(* Logix 5000 project; controller Drives_Line1 1756-L72 rev 20.13; software revision 20.04; part 16 of 21 *)
(* tags used below, declared in another part *)
   Exit_Accu_FBCounts_mm : DINT;
   Exit_Accu_Rev_mm : REAL;
   IO_State_Exit_Accu : INT;
   IO_State_Tmp_Exit_Accu : INT;
   ons : BOOL[32];
   TofReset : TIMER;
   TonNoResponse : TIMER;
   TonRefOn : TIMER;
   TonTensionOnSp : TIMER;
   zExit_Accu_EncCounts : DINT;
   zExit_Accu_Kp_Preg : REAL;
   zExit_Accu_Kp_Treg : REAL;
   zExit_Accu_MaxAccDec : REAL;
   zExit_Accu_NrOfCyl : DINT;
   zExit_Accu_Pos_PreLim : REAL;
   zExit_Accu_SpdRegMax : REAL;
   zExit_Accu_SpdRegMin : REAL;
   zExit_Accu_SpdTrim_HL : REAL;
   zExit_Accu_SpdtRim_LL : REAL;
   zExit_Accu_WLD_Preg : REAL;
   zExit_Accu_WLD_Treg : REAL;
   zNoMaster : BOOL;
   zTM3_Tens_Offset : REAL;
   Bridle_04 : UDT_Bridle_3M;
   EntryConfig : UDT_Config_Zone;
   Exit_Accu : UDT_Exit_Accu;
   ExitConfig : UDT_Config_Zone;
   ExitCtrl : UDT_Control_Zone;
   ExitStat : UDT_Status_Zone;
   In_Commands : UDT_Commands;
   In_Config : UDT_Config;
   In_Setpoints : UDT_Setpoints;
   LineCmd : UDT_Commands_Line;
   LineCtrl : UDT_Control_Line;
   LineStat : UDT_Status_Line;
   TM3 : UDT_TM;
(* P18_Exit_Accu, continued *)

ROUTINE R01_From_Master   (* ladder *)
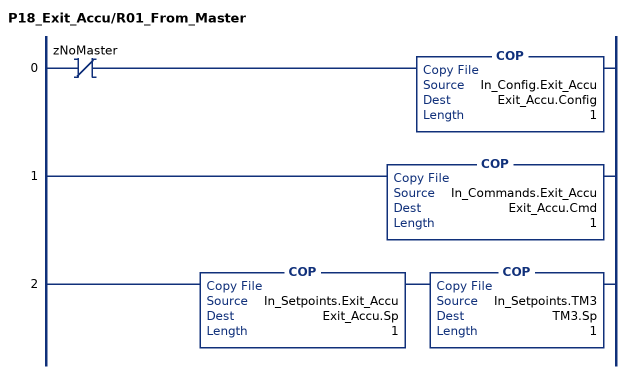
   0: XIO(zNoMaster)COP(In_Config.Exit_Accu,Exit_Accu.Config,1);
   1: COP(In_Commands.Exit_Accu,Exit_Accu.Cmd,1);
   2: COP(In_Setpoints.Exit_Accu,Exit_Accu.Sp,1)COP(In_Setpoints.TM3,TM3.Sp,1);
END_ROUTINE

ROUTINE R02_From_Drive   (* ladder *)
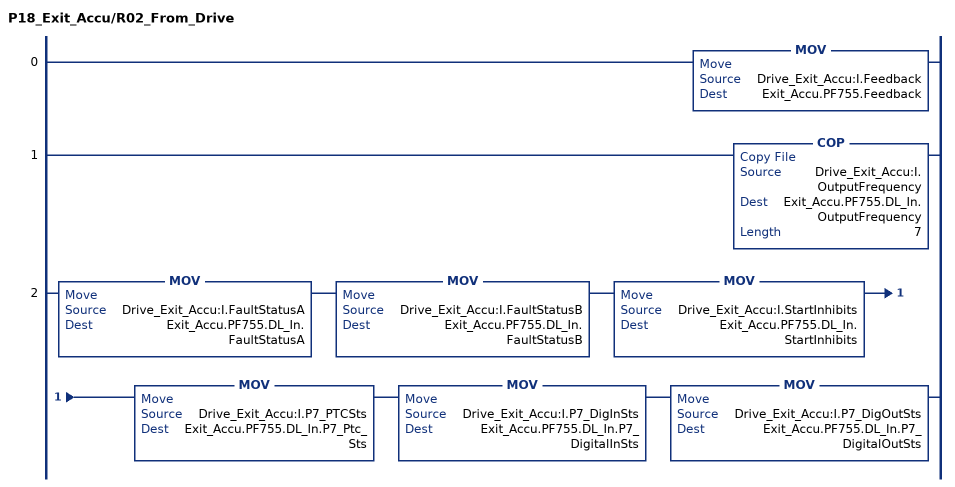
   0: MOV(Drive_Exit_Accu:I.Feedback,Exit_Accu.PF755.Feedback);
   1: COP(Drive_Exit_Accu:I.OutputFrequency,Exit_Accu.PF755.DL_In.OutputFrequency,7);
   2: MOV(Drive_Exit_Accu:I.FaultStatusA,Exit_Accu.PF755.DL_In.FaultStatusA)MOV(Drive_Exit_Accu:I.FaultStatusB,Exit_Accu.PF755.DL_In.FaultStatusB)MOV(Drive_Exit_Accu:I.StartInhibits,Exit_Accu.PF755.DL_In.StartInhibits)MOV(Drive_Exit_Accu:I.P7_PTCSts,Exit_Accu.PF755.DL_In.P7_Ptc_Sts)MOV(Drive_Exit_Accu:I.P7_DigInSts,Exit_Accu.PF755.DL_In.P7_DigitalInSts)MOV(Drive_Exit_Accu:I.P7_DigOutSts,Exit_Accu.PF755.DL_In.P7_DigitalOutSts);
END_ROUTINE

ROUTINE R03_Drive_Interface   (* ladder *)
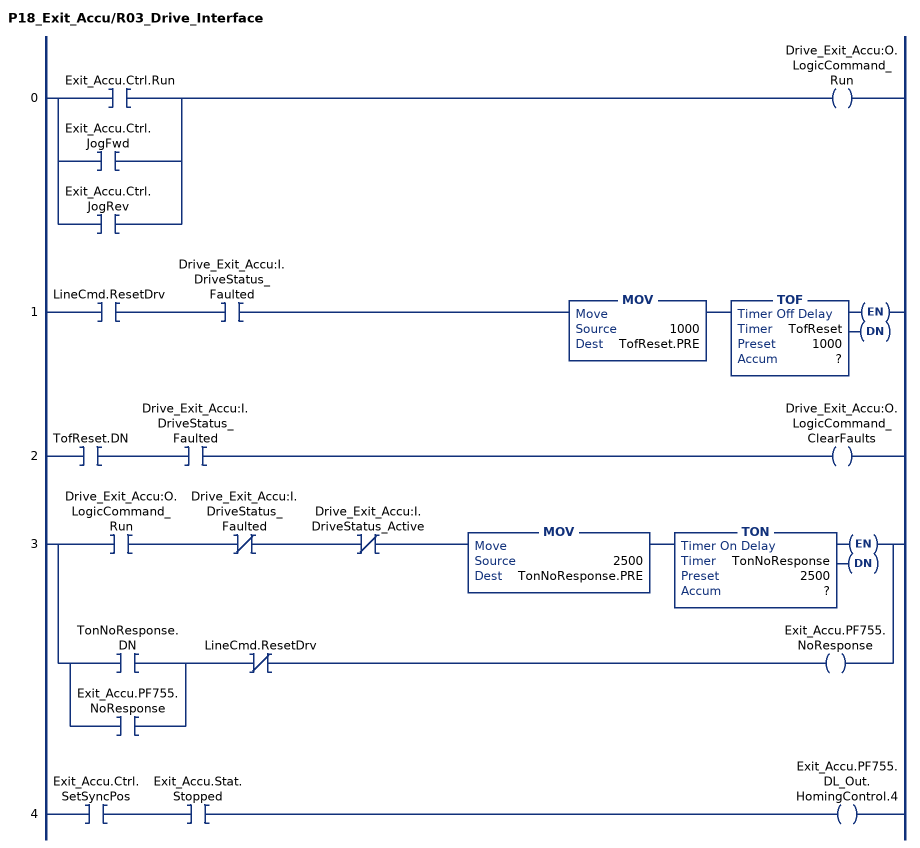
   0: [XIC(Exit_Accu.Ctrl.Run) ,XIC(Exit_Accu.Ctrl.JogFwd) ,XIC(Exit_Accu.Ctrl.JogRev) ]OTE(Drive_Exit_Accu:O.LogicCommand_Run);
   1: XIC(LineCmd.ResetDrv)XIC(Drive_Exit_Accu:I.DriveStatus_Faulted)MOV(1000,TofReset.PRE)TOF(TofReset,?,?);
   2: XIC(TofReset.DN)XIC(Drive_Exit_Accu:I.DriveStatus_Faulted)OTE(Drive_Exit_Accu:O.LogicCommand_ClearFaults);
   3: [XIC(Drive_Exit_Accu:O.LogicCommand_Run) XIO(Drive_Exit_Accu:I.DriveStatus_Faulted) XIO(Drive_Exit_Accu:I.DriveStatus_Active) MOV(2500,TonNoResponse.PRE) TON(TonNoResponse,?,?) ,[XIC(TonNoResponse.DN) ,XIC(Exit_Accu.PF755.NoResponse) ] XIO(LineCmd.ResetDrv) OTE(Exit_Accu.PF755.NoResponse) ];
   4: XIC(Exit_Accu.Ctrl.SetSyncPos)XIC(Exit_Accu.Stat.Stopped)OTE(Exit_Accu.PF755.DL_Out.HomingControl.4);
END_ROUTINE

ROUTINE R04_State   (* ladder *)
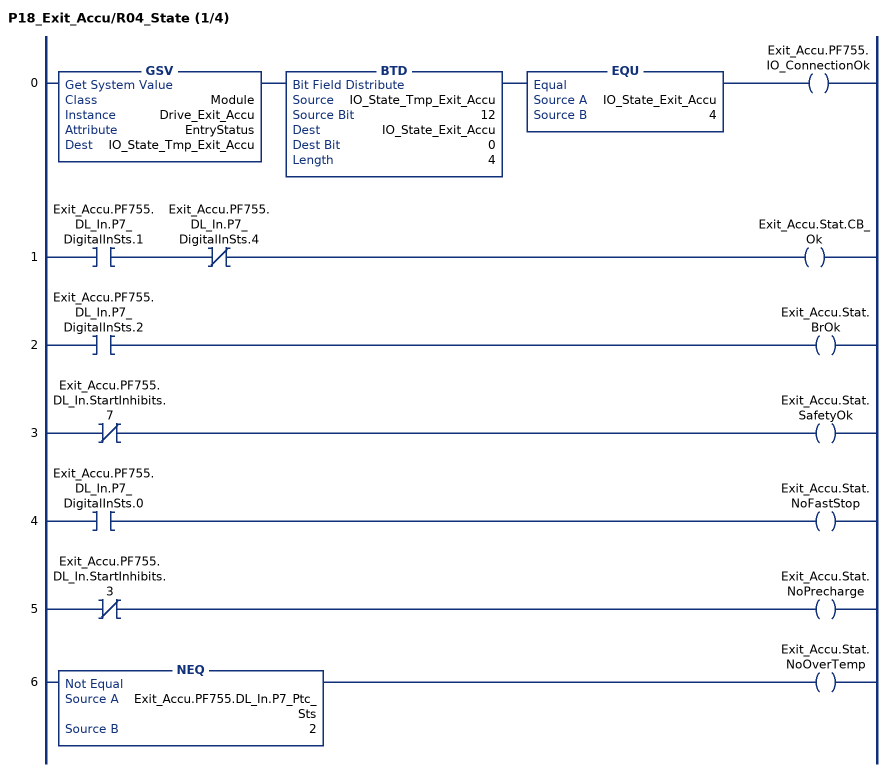
   0: GSV(Module,Drive_Exit_Accu,EntryStatus,IO_State_Tmp_Exit_Accu)BTD(IO_State_Tmp_Exit_Accu,12,IO_State_Exit_Accu,0,4)EQU(IO_State_Exit_Accu,4)OTE(Exit_Accu.PF755.IO_ConnectionOk);
   1: XIC(Exit_Accu.PF755.DL_In.P7_DigitalInSts.1)XIO(Exit_Accu.PF755.DL_In.P7_DigitalInSts.4)OTE(Exit_Accu.Stat.CB_Ok);
   2: XIC(Exit_Accu.PF755.DL_In.P7_DigitalInSts.2)OTE(Exit_Accu.Stat.BrOk);
   3: XIO(Exit_Accu.PF755.DL_In.StartInhibits.7)OTE(Exit_Accu.Stat.SafetyOk);
   4: XIC(Exit_Accu.PF755.DL_In.P7_DigitalInSts.0)OTE(Exit_Accu.Stat.NoFastStop);
   5: XIO(Exit_Accu.PF755.DL_In.StartInhibits.3)OTE(Exit_Accu.Stat.NoPrecharge);
   6: NEQ(Exit_Accu.PF755.DL_In.P7_Ptc_Sts,2)OTE(Exit_Accu.Stat.NoOverTemp);
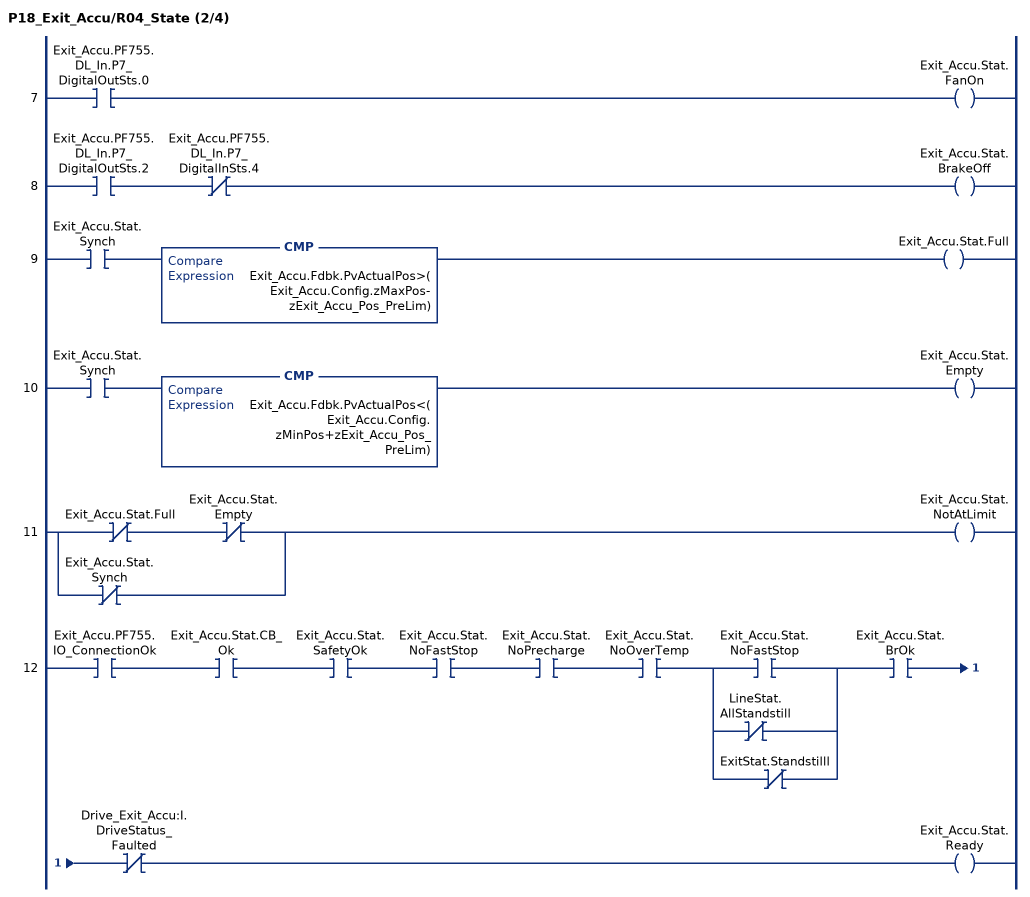
   7: XIC(Exit_Accu.PF755.DL_In.P7_DigitalOutSts.0)OTE(Exit_Accu.Stat.FanOn);
   8: XIC(Exit_Accu.PF755.DL_In.P7_DigitalOutSts.2)XIO(Exit_Accu.PF755.DL_In.P7_DigitalInSts.4)OTE(Exit_Accu.Stat.BrakeOff);
   9: XIC(Exit_Accu.Stat.Synch)CMP(Exit_Accu.Fdbk.PvActualPos>(Exit_Accu.Config.zMaxPos-zExit_Accu_Pos_PreLim))OTE(Exit_Accu.Stat.Full);
   10: XIC(Exit_Accu.Stat.Synch)CMP(Exit_Accu.Fdbk.PvActualPos<(Exit_Accu.Config.zMinPos+zExit_Accu_Pos_PreLim))OTE(Exit_Accu.Stat.Empty);
   11: [XIO(Exit_Accu.Stat.Full) XIO(Exit_Accu.Stat.Empty) ,XIO(Exit_Accu.Stat.Synch) ]OTE(Exit_Accu.Stat.NotAtLimit);
   12: XIC(Exit_Accu.PF755.IO_ConnectionOk)XIC(Exit_Accu.Stat.CB_Ok)XIC(Exit_Accu.Stat.SafetyOk)XIC(Exit_Accu.Stat.NoFastStop)XIC(Exit_Accu.Stat.NoPrecharge)XIC(Exit_Accu.Stat.NoOverTemp)[XIC(Exit_Accu.Stat.NoFastStop) ,XIO(LineStat.AllStandstill) ,XIO(ExitStat.Standstilll) ]XIC(Exit_Accu.Stat.BrOk)XIO(Drive_Exit_Accu:I.DriveStatus_Faulted)OTE(Exit_Accu.Stat.Ready);
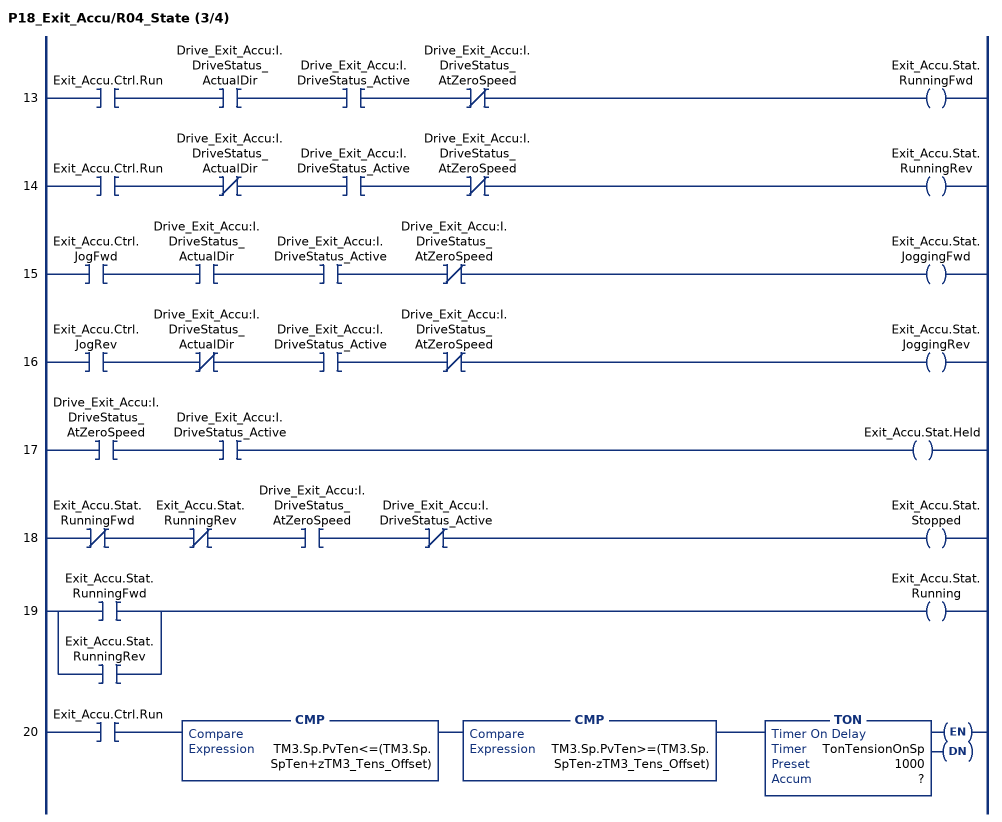
   13: XIC(Exit_Accu.Ctrl.Run)XIC(Drive_Exit_Accu:I.DriveStatus_ActualDir)XIC(Drive_Exit_Accu:I.DriveStatus_Active)XIO(Drive_Exit_Accu:I.DriveStatus_AtZeroSpeed)OTE(Exit_Accu.Stat.RunningFwd);
   14: XIC(Exit_Accu.Ctrl.Run)XIO(Drive_Exit_Accu:I.DriveStatus_ActualDir)XIC(Drive_Exit_Accu:I.DriveStatus_Active)XIO(Drive_Exit_Accu:I.DriveStatus_AtZeroSpeed)OTE(Exit_Accu.Stat.RunningRev);
   15: XIC(Exit_Accu.Ctrl.JogFwd)XIC(Drive_Exit_Accu:I.DriveStatus_ActualDir)XIC(Drive_Exit_Accu:I.DriveStatus_Active)XIO(Drive_Exit_Accu:I.DriveStatus_AtZeroSpeed)OTE(Exit_Accu.Stat.JoggingFwd);
   16: XIC(Exit_Accu.Ctrl.JogRev)XIO(Drive_Exit_Accu:I.DriveStatus_ActualDir)XIC(Drive_Exit_Accu:I.DriveStatus_Active)XIO(Drive_Exit_Accu:I.DriveStatus_AtZeroSpeed)OTE(Exit_Accu.Stat.JoggingRev);
   17: XIC(Drive_Exit_Accu:I.DriveStatus_AtZeroSpeed)XIC(Drive_Exit_Accu:I.DriveStatus_Active)OTE(Exit_Accu.Stat.Held);
   18: XIO(Exit_Accu.Stat.RunningFwd)XIO(Exit_Accu.Stat.RunningRev)XIC(Drive_Exit_Accu:I.DriveStatus_AtZeroSpeed)XIO(Drive_Exit_Accu:I.DriveStatus_Active)OTE(Exit_Accu.Stat.Stopped);
   19: [XIC(Exit_Accu.Stat.RunningFwd) ,XIC(Exit_Accu.Stat.RunningRev) ]OTE(Exit_Accu.Stat.Running);
   20: XIC(Exit_Accu.Ctrl.Run)CMP(TM3.Sp.PvTen<=(TM3.Sp.SpTen+zTM3_Tens_Offset))CMP(TM3.Sp.PvTen>=(TM3.Sp.SpTen-zTM3_Tens_Offset))TON(TonTensionOnSp,?,?);
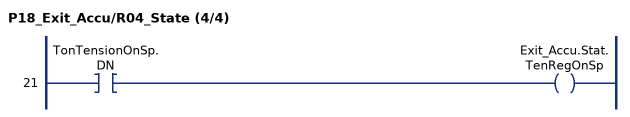
   21: XIC(TonTensionOnSp.DN)OTE(Exit_Accu.Stat.TenRegOnSp);
END_ROUTINE

ROUTINE R05_Control   (* ladder *)
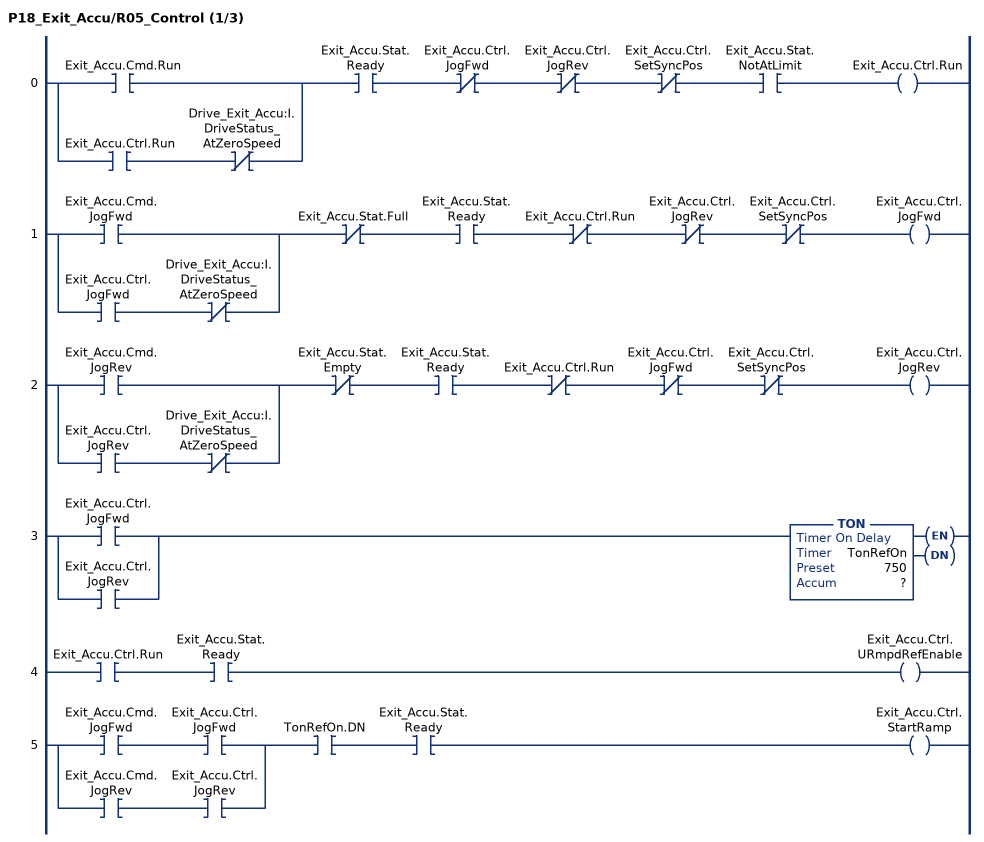
   0: [XIC(Exit_Accu.Cmd.Run) ,XIC(Exit_Accu.Ctrl.Run) XIO(Drive_Exit_Accu:I.DriveStatus_AtZeroSpeed) ]XIC(Exit_Accu.Stat.Ready)XIO(Exit_Accu.Ctrl.JogFwd)XIO(Exit_Accu.Ctrl.JogRev)XIO(Exit_Accu.Ctrl.SetSyncPos)XIC(Exit_Accu.Stat.NotAtLimit)OTE(Exit_Accu.Ctrl.Run);
   1: [XIC(Exit_Accu.Cmd.JogFwd) ,XIC(Exit_Accu.Ctrl.JogFwd) XIO(Drive_Exit_Accu:I.DriveStatus_AtZeroSpeed) ]XIO(Exit_Accu.Stat.Full)XIC(Exit_Accu.Stat.Ready)XIO(Exit_Accu.Ctrl.Run)XIO(Exit_Accu.Ctrl.JogRev)XIO(Exit_Accu.Ctrl.SetSyncPos)OTE(Exit_Accu.Ctrl.JogFwd);
   2: [XIC(Exit_Accu.Cmd.JogRev) ,XIC(Exit_Accu.Ctrl.JogRev) XIO(Drive_Exit_Accu:I.DriveStatus_AtZeroSpeed) ]XIO(Exit_Accu.Stat.Empty)XIC(Exit_Accu.Stat.Ready)XIO(Exit_Accu.Ctrl.Run)XIO(Exit_Accu.Ctrl.JogFwd)XIO(Exit_Accu.Ctrl.SetSyncPos)OTE(Exit_Accu.Ctrl.JogRev);
   3: [XIC(Exit_Accu.Ctrl.JogFwd) ,XIC(Exit_Accu.Ctrl.JogRev) ]TON(TonRefOn,?,?);
   4: XIC(Exit_Accu.Ctrl.Run)XIC(Exit_Accu.Stat.Ready)OTE(Exit_Accu.Ctrl.URmpdRefEnable);
   5: [XIC(Exit_Accu.Cmd.JogFwd) XIC(Exit_Accu.Ctrl.JogFwd) ,XIC(Exit_Accu.Cmd.JogRev) XIC(Exit_Accu.Ctrl.JogRev) ]XIC(TonRefOn.DN)XIC(Exit_Accu.Stat.Ready)OTE(Exit_Accu.Ctrl.StartRamp);
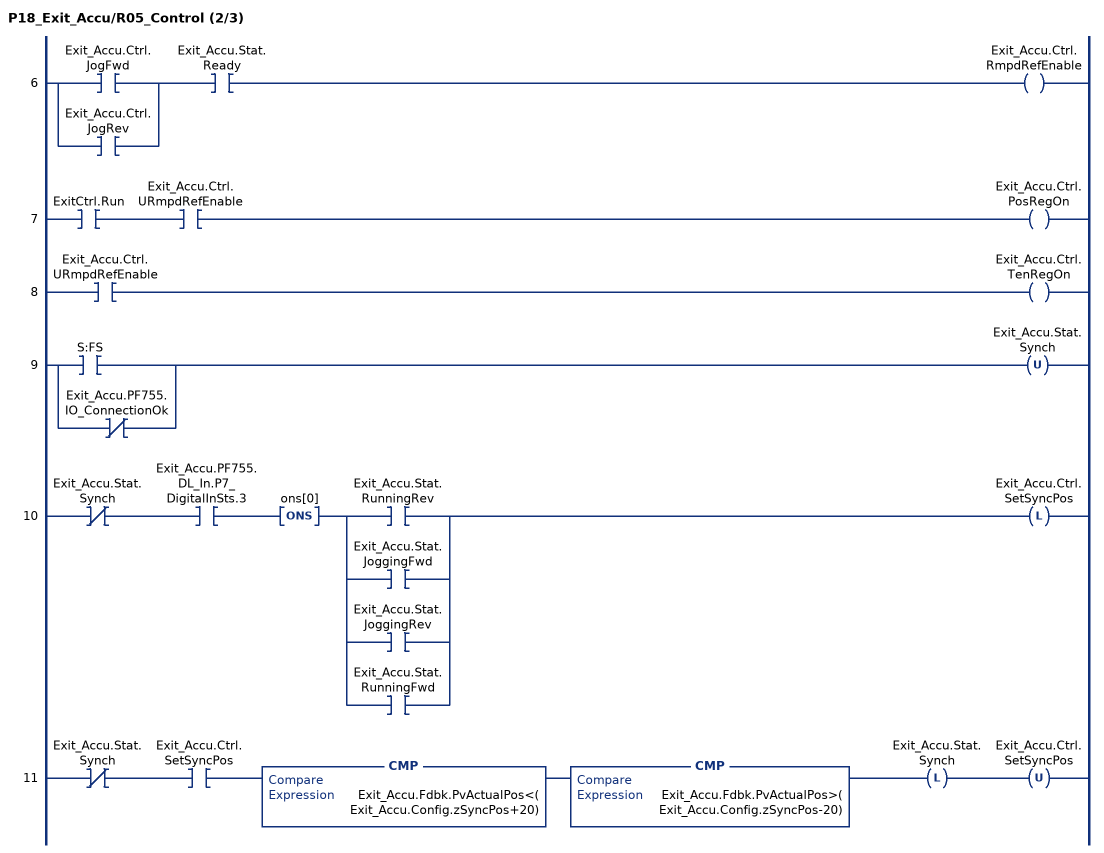
   6: [XIC(Exit_Accu.Ctrl.JogFwd) ,XIC(Exit_Accu.Ctrl.JogRev) ]XIC(Exit_Accu.Stat.Ready)OTE(Exit_Accu.Ctrl.RmpdRefEnable);
   7: XIC(ExitCtrl.Run)XIC(Exit_Accu.Ctrl.URmpdRefEnable)OTE(Exit_Accu.Ctrl.PosRegOn);
   8: XIC(Exit_Accu.Ctrl.URmpdRefEnable)OTE(Exit_Accu.Ctrl.TenRegOn);
   9: [XIC(S:FS) ,XIO(Exit_Accu.PF755.IO_ConnectionOk) ]OTU(Exit_Accu.Stat.Synch);
   10: XIO(Exit_Accu.Stat.Synch)XIC(Exit_Accu.PF755.DL_In.P7_DigitalInSts.3)ONS(ons[0])[XIC(Exit_Accu.Stat.RunningRev) ,XIC(Exit_Accu.Stat.JoggingFwd) ,XIC(Exit_Accu.Stat.JoggingRev) ,XIC(Exit_Accu.Stat.RunningFwd) ]OTL(Exit_Accu.Ctrl.SetSyncPos);
   11: XIO(Exit_Accu.Stat.Synch)XIC(Exit_Accu.Ctrl.SetSyncPos)CMP(Exit_Accu.Fdbk.PvActualPos<(Exit_Accu.Config.zSyncPos+20))CMP(Exit_Accu.Fdbk.PvActualPos>(Exit_Accu.Config.zSyncPos-20))OTL(Exit_Accu.Stat.Synch)OTU(Exit_Accu.Ctrl.SetSyncPos);
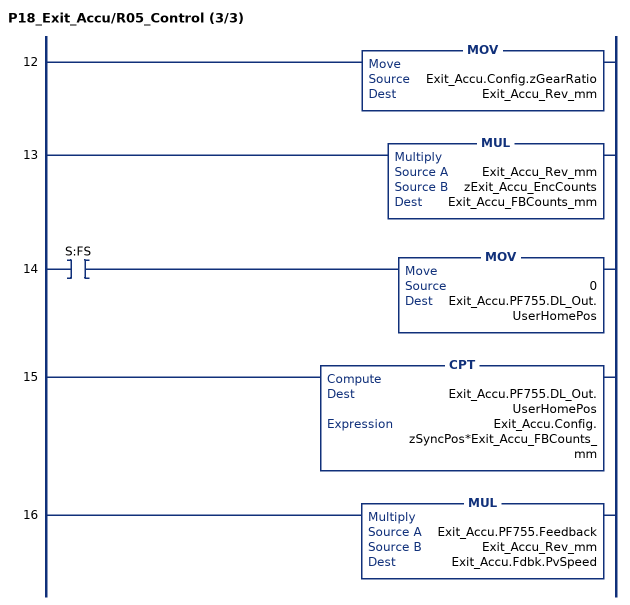
   12: MOV(Exit_Accu.Config.zGearRatio,Exit_Accu_Rev_mm);
   13: MUL(Exit_Accu_Rev_mm,zExit_Accu_EncCounts,Exit_Accu_FBCounts_mm);
   14: XIC(S:FS)MOV(0,Exit_Accu.PF755.DL_Out.UserHomePos);
   15: CPT(Exit_Accu.PF755.DL_Out.UserHomePos,Exit_Accu.Config.zSyncPos*Exit_Accu_FBCounts_mm);
   16: MUL(Exit_Accu.PF755.Feedback,Exit_Accu_Rev_mm,Exit_Accu.Fdbk.PvSpeed);
END_ROUTINE

ROUTINE R10_TenReg   (* function block diagram *)
   SHEET 1   // Scale setpoint
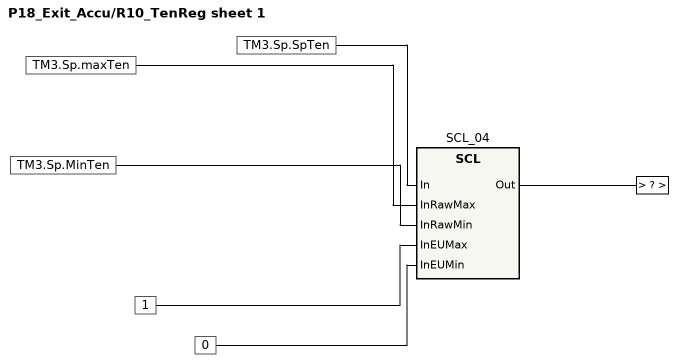
   SCL_04 : SCL(In := TM3.Sp.SpTen, InRawMax := TM3.Sp.maxTen, InRawMin := TM3.Sp.MinTen, InEUMax := 1, InEUMin := 0);
   WIRE(?) := SCL_04.Out;
   SHEET 2   // Scale tension feedback
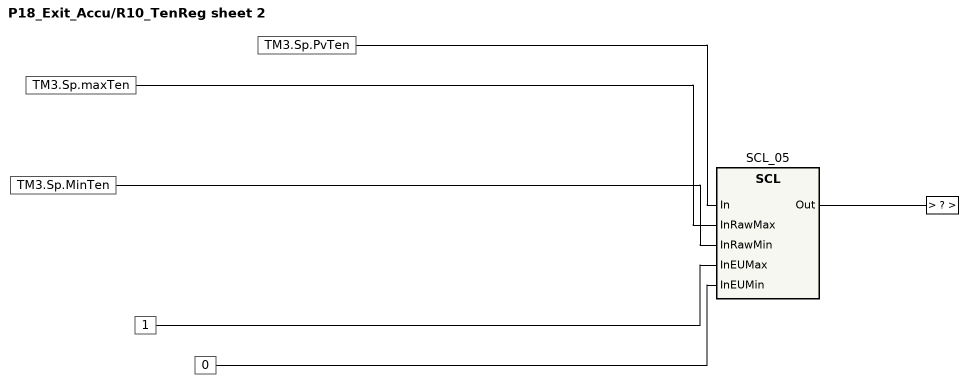
   SCL_05 : SCL(In := TM3.Sp.PvTen, InRawMax := TM3.Sp.maxTen, InRawMin := TM3.Sp.MinTen, InEUMax := 1, InEUMin := 0);
   WIRE(?) := SCL_05.Out;
   SHEET 3   // Trim limits
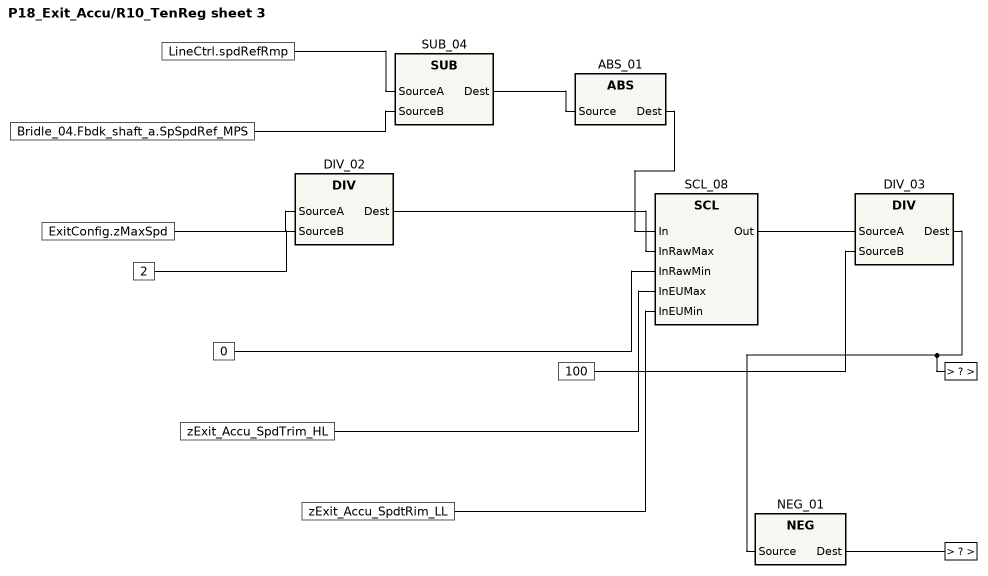
   DIV_02 : DIV(SourceA := ExitConfig.zMaxSpd, SourceB := 2);
   SUB_04 : SUB(SourceA := LineCtrl.spdRefRmp, SourceB := Bridle_04.Fbdk_shaft_a.SpSpdRef_MPS);
   ABS_01 : ABS(Source := SUB_04.Dest);
   SCL_08 : SCL(In := ABS_01.Dest, InRawMax := DIV_02.Dest, InRawMin := 0, InEUMax := zExit_Accu_SpdTrim_HL, InEUMin := zExit_Accu_SpdtRim_LL);
   DIV_03 : DIV(SourceA := SCL_08.Out, SourceB := 100);
   NEG_01 : NEG(Source := DIV_03.Dest);
   WIRE(?) := DIV_03.Dest;
   WIRE(?) := NEG_01.Dest;
   SHEET 4   // Tension regulator
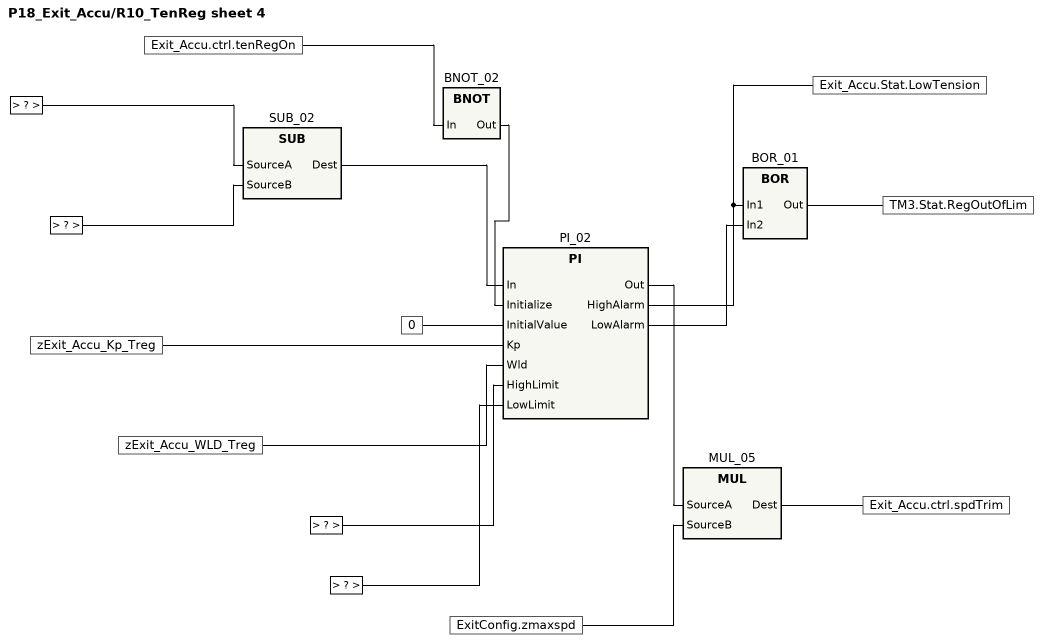
   SUB_02 : SUB(SourceA := WIRE(?), SourceB := WIRE(?));
   BNOT_02 : BNOT(In := Exit_Accu.ctrl.tenRegOn);
   PI_02 : PI(In := SUB_02.Dest, Initialize := BNOT_02.Out, InitialValue := 0, Kp := zExit_Accu_Kp_Treg, Wld := zExit_Accu_WLD_Treg, HighLimit := WIRE(?), LowLimit := WIRE(?));
   MUL_05 : MUL(SourceA := PI_02.Out, SourceB := ExitConfig.zmaxspd);
   BOR_01 : BOR(In1 := PI_02.HighAlarm, In2 := PI_02.LowAlarm);
   Exit_Accu.Stat.LowTension := PI_02.HighAlarm;
   Exit_Accu.ctrl.spdTrim := MUL_05.Dest;
   TM3.Stat.RegOutOfLim := BOR_01.Out;
END_ROUTINE

ROUTINE R11_PosReg   (* function block diagram *)
   SHEET 1   // Scale feedback
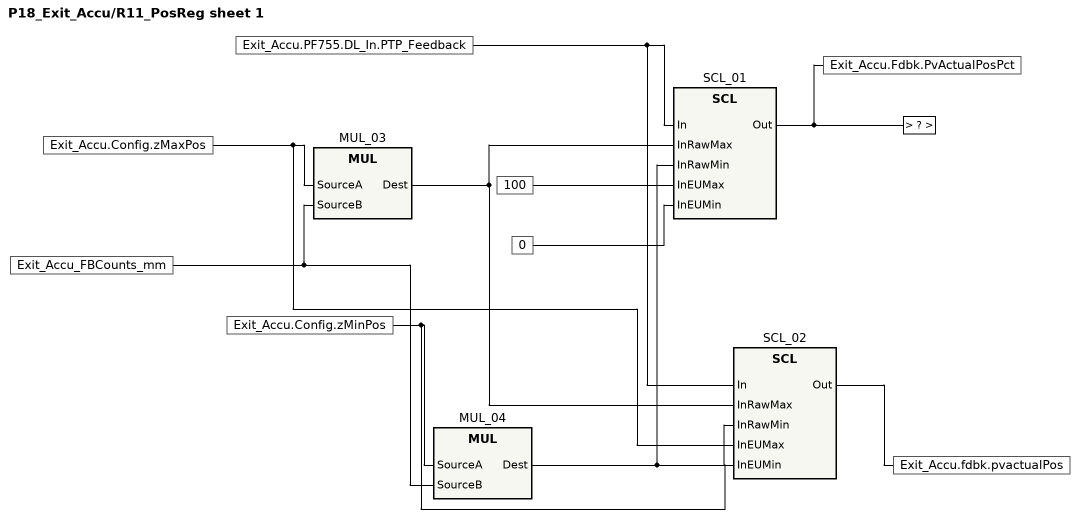
   MUL_03 : MUL(SourceA := Exit_Accu.Config.zMaxPos, SourceB := Exit_Accu_FBCounts_mm);
   MUL_04 : MUL(SourceA := Exit_Accu.Config.zMinPos, SourceB := Exit_Accu_FBCounts_mm);
   SCL_01 : SCL(In := Exit_Accu.PF755.DL_In.PTP_Feedback, InRawMax := MUL_03.Dest, InRawMin := MUL_04.Dest, InEUMax := 100, InEUMin := 0);
   SCL_02 : SCL(In := Exit_Accu.PF755.DL_In.PTP_Feedback, InRawMax := MUL_03.Dest, InRawMin := MUL_04.Dest, InEUMax := Exit_Accu.Config.zMaxPos, InEUMin := Exit_Accu.Config.zMinPos);
   Exit_Accu.Fdbk.PvActualPosPct := SCL_01.Out;
   Exit_Accu.fdbk.pvactualPos := SCL_02.Out;
   WIRE(?) := SCL_01.Out;
   SHEET 2   // Position regulator
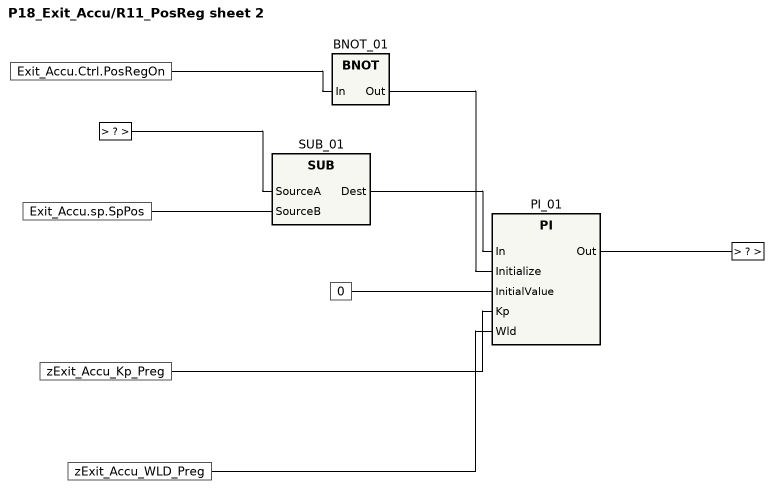
   BNOT_01 : BNOT(In := Exit_Accu.Ctrl.PosRegOn);
   SUB_01 : SUB(SourceA := WIRE(?), SourceB := Exit_Accu.sp.SpPos);
   PI_01 : PI(In := SUB_01.Dest, Initialize := BNOT_01.Out, InitialValue := 0, Kp := zExit_Accu_Kp_Preg, Wld := zExit_Accu_WLD_Preg);
   WIRE(?) := PI_01.Out;
   SHEET 3   // Scale position regulator output
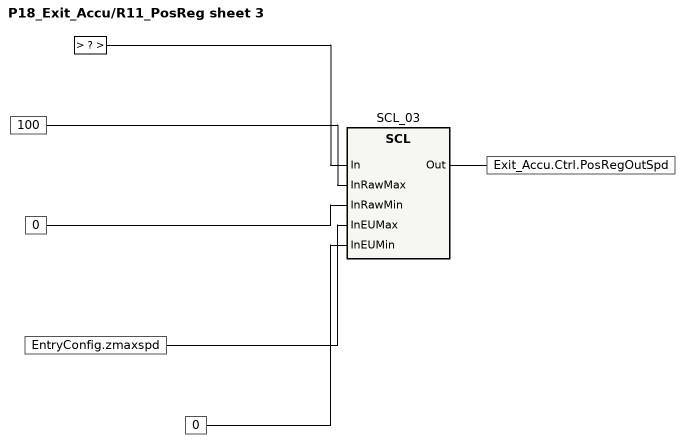
   SCL_03 : SCL(In := WIRE(?), InRawMax := 100, InRawMin := 0, InEUMax := EntryConfig.zmaxspd, InEUMin := 0);
   Exit_Accu.Ctrl.PosRegOutSpd := SCL_03.Out;
END_ROUTINE

ROUTINE R12_DriveRef   (* function block diagram *)
   SHEET 1   // Speed reference selection
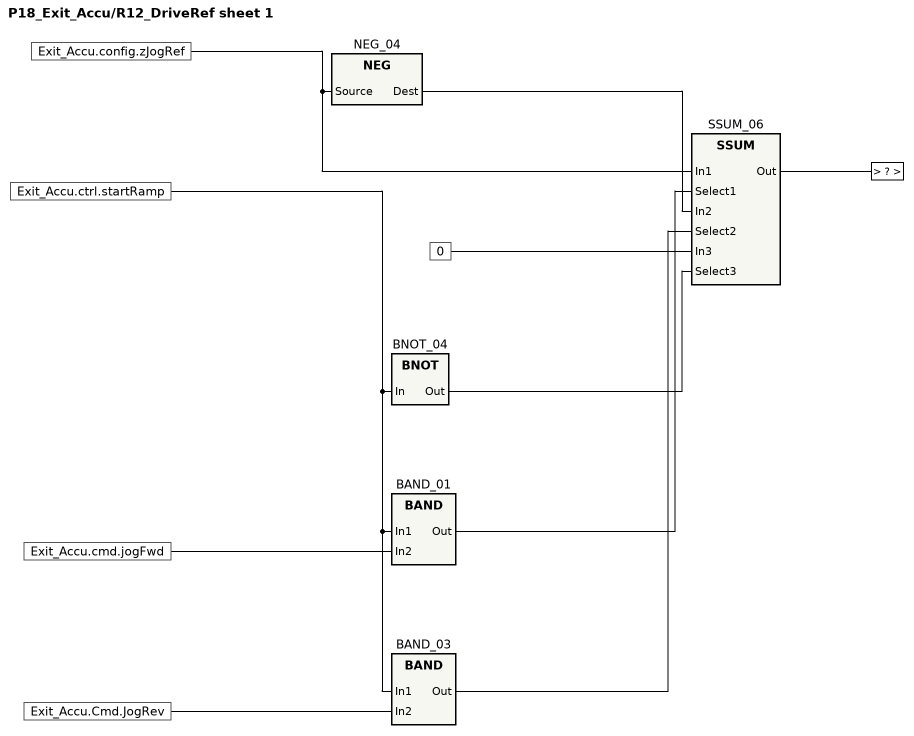
   NEG_04 : NEG(Source := Exit_Accu.config.zJogRef);
   BNOT_04 : BNOT(In := Exit_Accu.ctrl.startRamp);
   BAND_01 : BAND(In1 := Exit_Accu.ctrl.startRamp, In2 := Exit_Accu.cmd.jogFwd);
   BAND_03 : BAND(In1 := Exit_Accu.ctrl.startRamp, In2 := Exit_Accu.Cmd.JogRev);
   SSUM_06 : SSUM(In1 := Exit_Accu.config.zJogRef, Select1 := BAND_01.Out, In2 := NEG_04.Dest, Select2 := BAND_03.Out, In3 := 0, Select3 := BNOT_04.Out);
   WIRE(?) := SSUM_06.Out;
   SHEET 2   // S-Curve
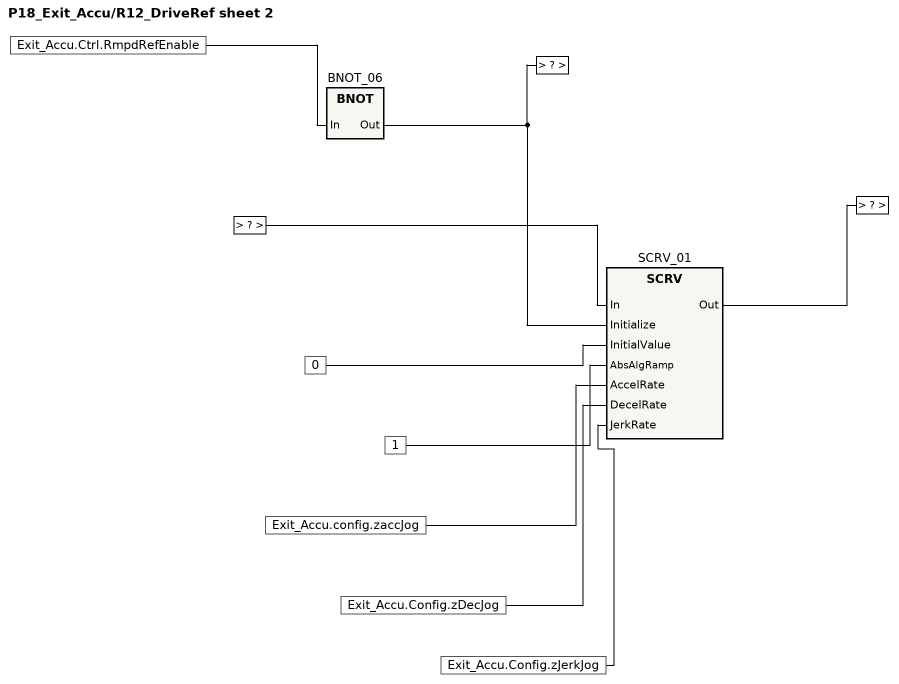
   BNOT_06 : BNOT(In := Exit_Accu.Ctrl.RmpdRefEnable);
   WIRE(?) := BNOT_06.Out;
   SCRV_01 : SCRV(In := WIRE(?), Initialize := BNOT_06.Out, InitialValue := 0, AbsAlgRamp := 1, AccelRate := Exit_Accu.config.zaccJog, DecelRate := Exit_Accu.Config.zDecJog, JerkRate := Exit_Accu.Config.zJerkJog);
   WIRE(?) := SCRV_01.Out;
   SHEET 3   // Run speed reference (Vp - Vx)
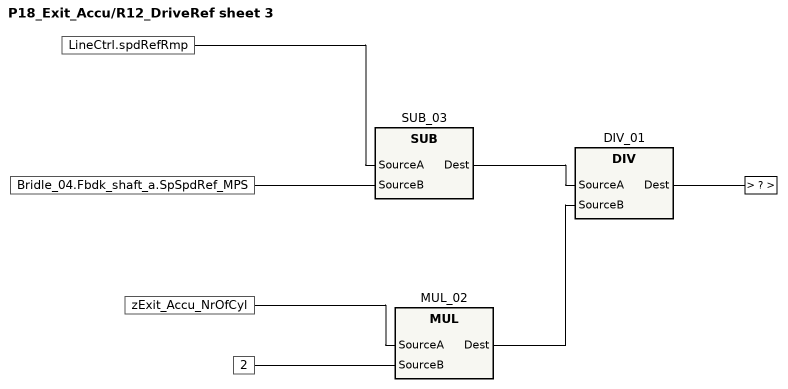
   SUB_03 : SUB(SourceA := LineCtrl.spdRefRmp, SourceB := Bridle_04.Fbdk_shaft_a.SpSpdRef_MPS);
   MUL_02 : MUL(SourceA := zExit_Accu_NrOfCyl, SourceB := 2);
   DIV_01 : DIV(SourceA := SUB_03.Dest, SourceB := MUL_02.Dest);
   WIRE(?) := DIV_01.Dest;
   SHEET 4   // Select ramped/unramped reference
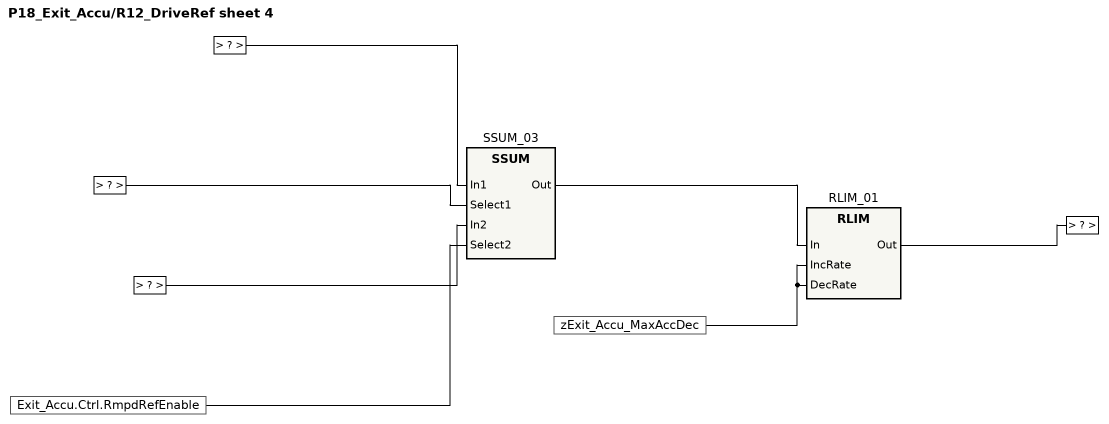
   SSUM_03 : SSUM(In1 := WIRE(?), Select1 := WIRE(?), In2 := WIRE(?), Select2 := Exit_Accu.Ctrl.RmpdRefEnable);
   RLIM_01 : RLIM(In := SSUM_03.Out, IncRate := zExit_Accu_MaxAccDec, DecRate := zExit_Accu_MaxAccDec);
   WIRE(?) := RLIM_01.Out;
   SHEET 5   // Limit speed regulator
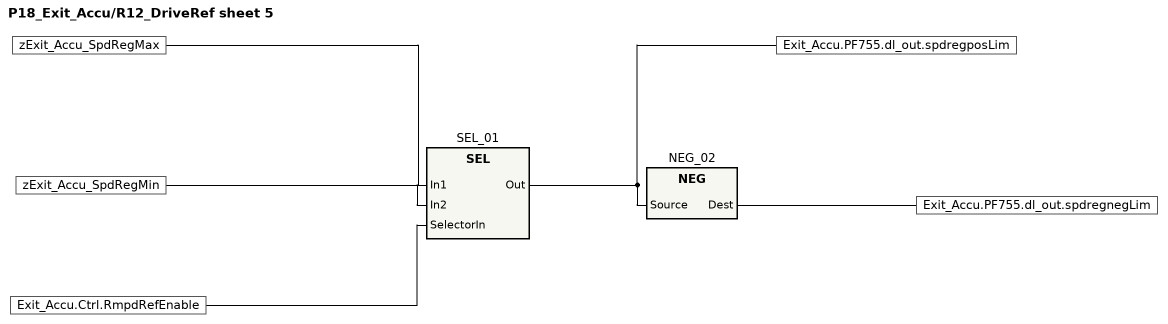
   SEL_01 : SEL(In1 := zExit_Accu_SpdRegMax, In2 := zExit_Accu_SpdRegMin, SelectorIn := Exit_Accu.Ctrl.RmpdRefEnable);
   NEG_02 : NEG(Source := SEL_01.Out);
   Exit_Accu.PF755.dl_out.spdregposLim := SEL_01.Out;
   Exit_Accu.PF755.dl_out.spdregnegLim := NEG_02.Dest;
   SHEET 6   // Final speed reference
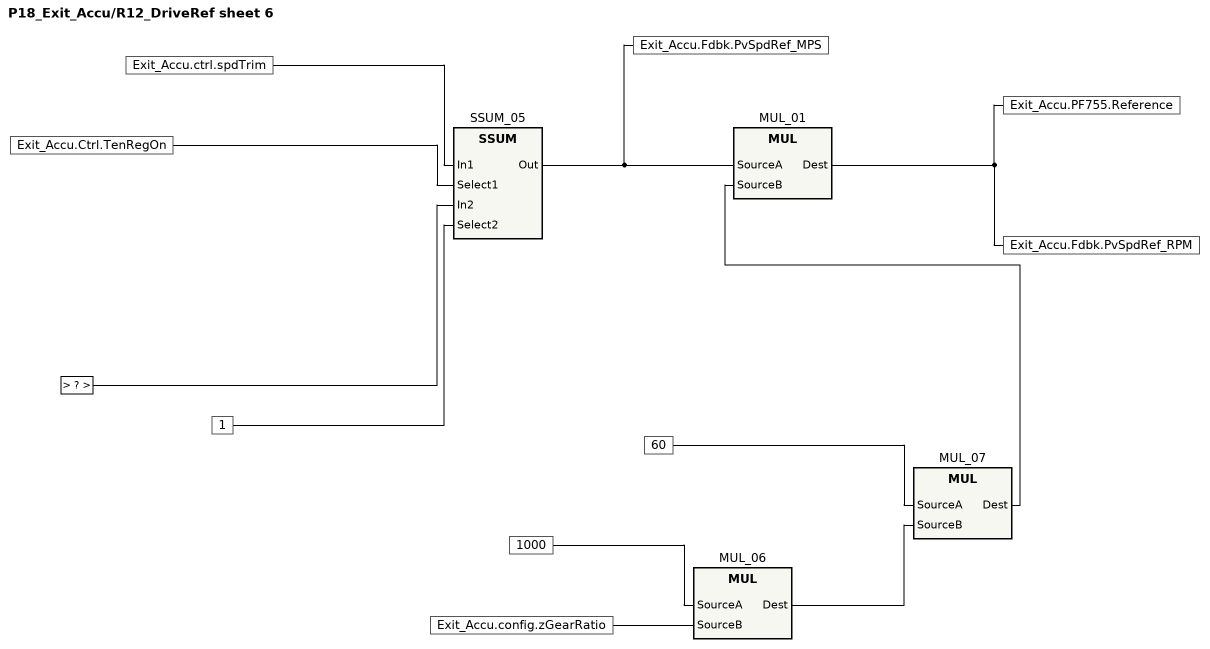
   SSUM_05 : SSUM(In1 := Exit_Accu.ctrl.spdTrim, Select1 := Exit_Accu.Ctrl.TenRegOn, In2 := WIRE(?), Select2 := 1);
   Exit_Accu.Fdbk.PvSpdRef_MPS := SSUM_05.Out;
   MUL_06 : MUL(SourceA := 1000, SourceB := Exit_Accu.config.zGearRatio);
   MUL_07 : MUL(SourceA := 60, SourceB := MUL_06.Dest);
   MUL_01 : MUL(SourceA := SSUM_05.Out, SourceB := MUL_07.Dest);
   Exit_Accu.PF755.Reference := MUL_01.Dest;
   Exit_Accu.Fdbk.PvSpdRef_RPM := MUL_01.Dest;
END_ROUTINE
